// TIA Portal V16 export
// export: Created 2022-11-14T17:35:32.0229208Z, ExportSetting WithDefaults, DisplayName Totally Integrated Automation Portal, DisplayVersion V16, DisplayName TIA Portal Version Control Interface, DisplayVersion V16, DisplayName TIA Portal Openness, DisplayVersion V16, DisplayName STEP 7 Professional, DisplayVersion V16, DisplayName STEP 7 Safety, DisplayVersion V16, DisplayName WinCC Advanced, DisplayVersion V16
FUNCTION "FC72_Conveyor_0_IN_1_OUT" : Void   // FC72, LAD
TITLE = Conveyor_0_IN_1_OUT
{ S7_Optimized_Access := 'FALSE' }
VERSION : 0.1
// stored: AutoNumber false, IsIECCheckEnabled false, SetENOAutomatically false, UDAEnableTagReadback false
   VAR_TEMP   // added for the SCL form of the ladder/FBD networks
      _w1 : Bool;
   END_VAR
BEGIN

REGION Network 1: Conveyor manual movement
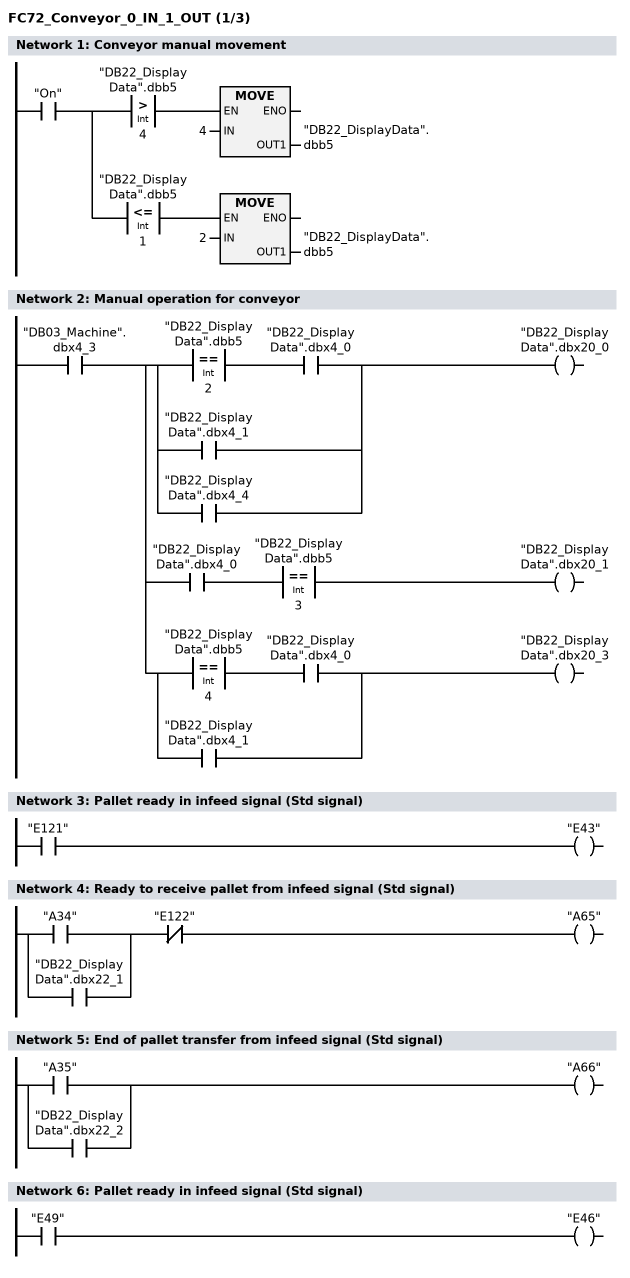
   RUNG wire#powerrail
      Contact( "On" )
      wire#w1
      { S7_Templates := "SrcType := Int" } GT_Contact(in1 := "DB22_DisplayData".dbb5, in2 := 4)
      { S7_GenerateENO := "TRUE" } Move(in := 4, out1 => "DB22_DisplayData".dbb5)
   END_RUNG
   RUNG wire#w1
      { S7_Templates := "SrcType := Int" } LE_Contact(in1 := "DB22_DisplayData".dbb5, in2 := 1)
      { S7_GenerateENO := "TRUE" } Move(in := 2, out1 => "DB22_DisplayData".dbb5)
   END_RUNG
   // the same network as SCL:
   IF "On" AND ("DB22_DisplayData".dbb5 > 4) THEN "DB22_DisplayData".dbb5 := 4; END_IF;
   IF "On" AND ("DB22_DisplayData".dbb5 <= 1) THEN "DB22_DisplayData".dbb5 := 2; END_IF;
END_REGION

REGION Network 2: Manual operation for conveyor
   RUNG wire#powerrail
      Contact( "DB03_Machine".dbx4_3 )
      wire#w1
      { S7_Templates := "SrcType := Int" } EQ_Contact(in1 := "DB22_DisplayData".dbb5, in2 := 2)
      Contact( "DB22_DisplayData".dbx4_0 )
      wire#w2
      Coil( "DB22_DisplayData".dbx20_0 )
   END_RUNG
   RUNG wire#w1
      Contact( "DB22_DisplayData".dbx4_1 )
   END_RUNG wire#w2
   RUNG wire#w1
      Contact( "DB22_DisplayData".dbx4_4 )
   END_RUNG wire#w2
   RUNG wire#w1
      Contact( "DB22_DisplayData".dbx4_0 )
      { S7_Templates := "SrcType := Int" } EQ_Contact(in1 := "DB22_DisplayData".dbb5, in2 := 3)
      Coil( "DB22_DisplayData".dbx20_1 )
   END_RUNG
   RUNG wire#w1
      { S7_Templates := "SrcType := Int" } EQ_Contact(in1 := "DB22_DisplayData".dbb5, in2 := 4)
      Contact( "DB22_DisplayData".dbx4_0 )
      wire#w3
      Coil( "DB22_DisplayData".dbx20_3 )
   END_RUNG
   RUNG wire#w1
      Contact( "DB22_DisplayData".dbx4_1 )
   END_RUNG wire#w3
   // the same network as SCL:
   "DB22_DisplayData".dbx20_0 := "DB03_Machine".dbx4_3 AND ((("DB22_DisplayData".dbb5 = 2) AND "DB22_DisplayData".dbx4_0) OR "DB22_DisplayData".dbx4_1 OR "DB22_DisplayData".dbx4_4);
   "DB22_DisplayData".dbx20_1 := "DB03_Machine".dbx4_3 AND "DB22_DisplayData".dbx4_0 AND ("DB22_DisplayData".dbb5 = 3);
   "DB22_DisplayData".dbx20_3 := "DB03_Machine".dbx4_3 AND ((("DB22_DisplayData".dbb5 = 4) AND "DB22_DisplayData".dbx4_0) OR "DB22_DisplayData".dbx4_1);
END_REGION

REGION Network 3: Pallet ready in infeed signal (Std signal)
   RUNG wire#powerrail
      Contact( "E121" )
      Coil( "E43" )
   END_RUNG
   // the same network as SCL:
   "E43" := "E121";
END_REGION

REGION Network 4: Ready to receive pallet from infeed signal (Std signal)
   RUNG wire#powerrail
      Contact( "A34" )
      wire#w1
      I_Contact( "E122" )
      Coil( "A65" )
   END_RUNG
   RUNG wire#powerrail
      Contact( "DB22_DisplayData".dbx22_1 )
   END_RUNG wire#w1
   // the same network as SCL:
   "A65" := ("A34" OR "DB22_DisplayData".dbx22_1) AND NOT "E122";
END_REGION

REGION Network 5: End of pallet transfer from infeed signal (Std signal)
   RUNG wire#powerrail
      Contact( "A35" )
      wire#w1
      Coil( "A66" )
   END_RUNG
   RUNG wire#powerrail
      Contact( "DB22_DisplayData".dbx22_2 )
   END_RUNG wire#w1
   // the same network as SCL:
   "A66" := "A35" OR "DB22_DisplayData".dbx22_2;
END_REGION

REGION Network 6: Pallet ready in infeed signal (Std signal)
   RUNG wire#powerrail
      Contact( "E49" )
      Coil( "E46" )
   END_RUNG
   // the same network as SCL:
   "E46" := "E49";
END_REGION

REGION Network 7: >>>>> OUTFEED CONVEYOR <<<<<<
END_REGION

REGION Network 8: Time for pallet unload with forklift
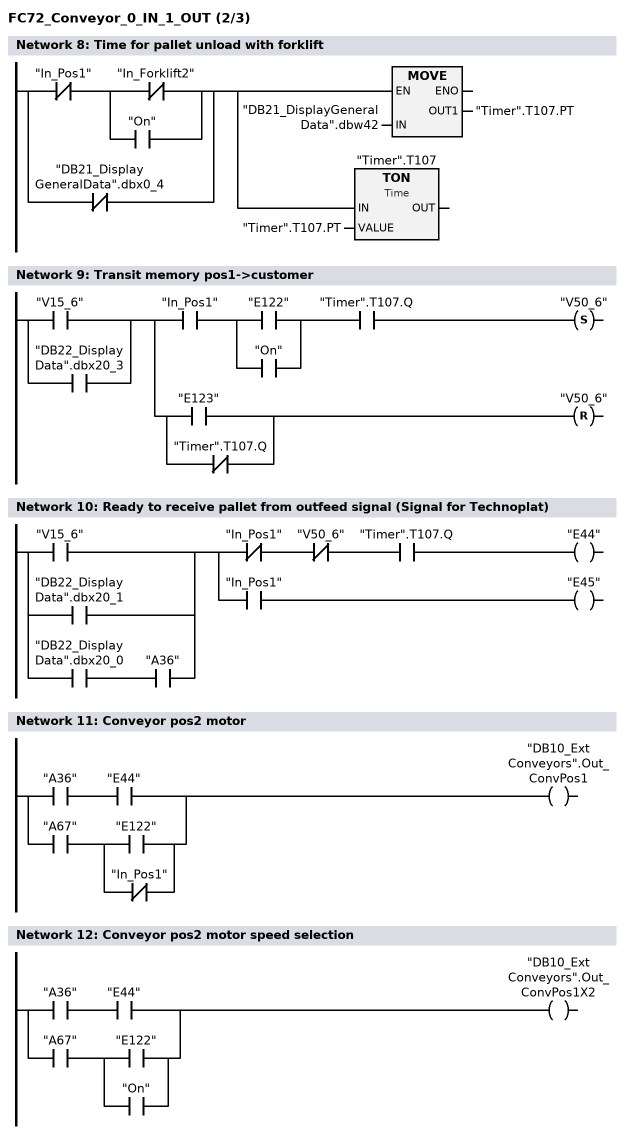
   #_w1 := (NOT "In_Pos1" AND (NOT "In_Forklift2" OR "On")) OR NOT "DB21_DisplayGeneralData".dbx0_4;
   IF #_w1 THEN "Timer".T107.PT := "DB21_DisplayGeneralData".dbw42; END_IF;
   "Timer".T107.TON(IN := #_w1, PT := "Timer".T107.PT);   // TON coil
END_REGION

REGION Network 9: Transit memory pos1->customer
   RUNG wire#powerrail
      Contact( "V15_6" )
      wire#w1
      Contact( "In_Pos1" )
      wire#w2
      Contact( "E122" )
      wire#w3
      Contact( "Timer".T107.Q )
      S_Coil( "V50_6" )
   END_RUNG
   RUNG wire#powerrail
      Contact( "DB22_DisplayData".dbx20_3 )
   END_RUNG wire#w1
   RUNG wire#w2
      Contact( "On" )
   END_RUNG wire#w3
   RUNG wire#w1
      Contact( "E123" )
      wire#w4
      R_Coil( "V50_6" )
   END_RUNG
   RUNG wire#w1
      I_Contact( "Timer".T107.Q )
   END_RUNG wire#w4
   // the same network as SCL:
   #_w1 := "V15_6" OR "DB22_DisplayData".dbx20_3;
   IF #_w1 AND "In_Pos1" AND ("E122" OR "On") AND "Timer".T107.Q THEN "V50_6" := TRUE; END_IF;
   IF #_w1 AND ("E123" OR NOT "Timer".T107.Q) THEN "V50_6" := FALSE; END_IF;
END_REGION

REGION Network 10: Ready to receive pallet from outfeed signal (Signal for Technoplat)
   RUNG wire#powerrail
      Contact( "V15_6" )
      wire#w1
      I_Contact( "In_Pos1" )
      I_Contact( "V50_6" )
      Contact( "Timer".T107.Q )
      Coil( "E44" )
   END_RUNG
   RUNG wire#powerrail
      Contact( "DB22_DisplayData".dbx20_1 )
   END_RUNG wire#w1
   RUNG wire#powerrail
      Contact( "DB22_DisplayData".dbx20_0 )
      Contact( "A36" )
   END_RUNG wire#w1
   RUNG wire#w1
      Contact( "In_Pos1" )
      Coil( "E45" )
   END_RUNG
   // the same network as SCL:
   #_w1 := "V15_6" OR "DB22_DisplayData".dbx20_1 OR ("DB22_DisplayData".dbx20_0 AND "A36");
   "E44" := #_w1 AND NOT "In_Pos1" AND NOT "V50_6" AND "Timer".T107.Q;
   "E45" := #_w1 AND "In_Pos1";
END_REGION

REGION Network 11: Conveyor pos2 motor
   RUNG wire#powerrail
      Contact( "A36" )
      Contact( "E44" )
      wire#w1
      Coil( "DB10_ExtConveyors".Out_ConvPos1 )
   END_RUNG
   RUNG wire#powerrail
      Contact( "A67" )
      wire#w2
      Contact( "E122" )
   END_RUNG wire#w1
   RUNG wire#w2
      I_Contact( "In_Pos1" )
   END_RUNG wire#w1
   // the same network as SCL:
   "DB10_ExtConveyors".Out_ConvPos1 := ("A36" AND "E44") OR ("A67" AND ("E122" OR NOT "In_Pos1"));
END_REGION

REGION Network 12: Conveyor pos2 motor speed selection
   RUNG wire#powerrail
      Contact( "A36" )
      Contact( "E44" )
      wire#w1
      Coil( "DB10_ExtConveyors".Out_ConvPos1X2 )
   END_RUNG
   RUNG wire#powerrail
      Contact( "A67" )
      wire#w2
      Contact( "E122" )
   END_RUNG wire#w1
   RUNG wire#w2
      Contact( "On" )
   END_RUNG wire#w1
   // the same network as SCL:
   "DB10_ExtConveyors".Out_ConvPos1X2 := ("A36" AND "E44") OR ("A67" AND ("E122" OR "On"));
END_REGION

REGION Network 13: Pallet ready in outfeed signal
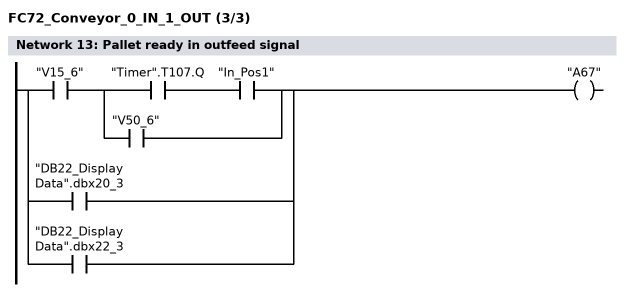
   RUNG wire#powerrail
      Contact( "V15_6" )
      wire#w1
      Contact( "Timer".T107.Q )
      Contact( "In_Pos1" )
      wire#w2
      Coil( "A67" )
   END_RUNG
   RUNG wire#w1
      Contact( "V50_6" )
   END_RUNG wire#w2
   RUNG wire#powerrail
      Contact( "DB22_DisplayData".dbx20_3 )
   END_RUNG wire#w2
   RUNG wire#powerrail
      Contact( "DB22_DisplayData".dbx22_3 )
   END_RUNG wire#w2
   // the same network as SCL:
   "A67" := ("V15_6" AND (("Timer".T107.Q AND "In_Pos1") OR "V50_6")) OR "DB22_DisplayData".dbx20_3 OR "DB22_DisplayData".dbx22_3;
END_REGION
END_FUNCTION
